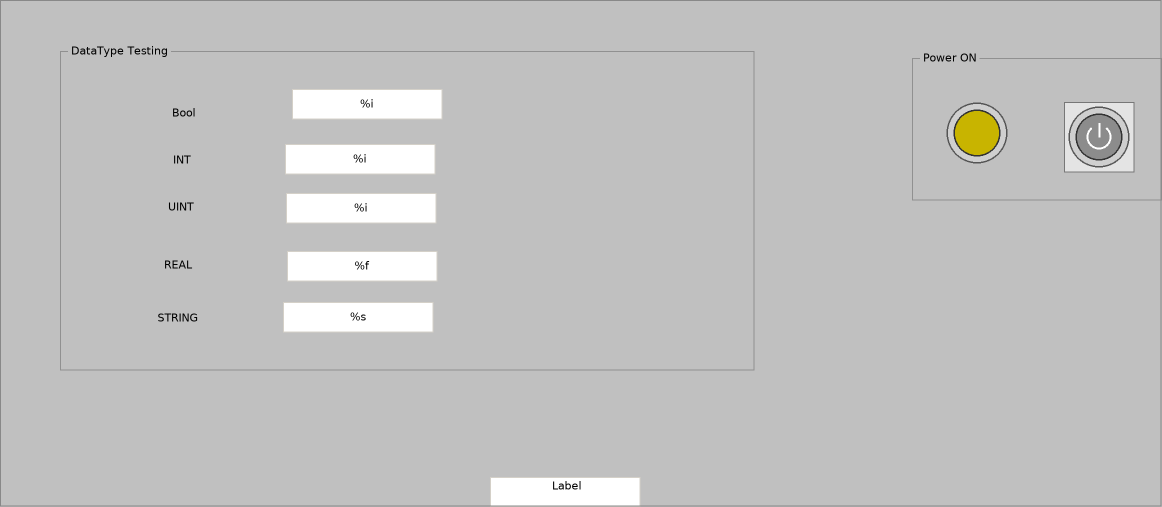
VISUALIZATION HMI  // 1162x507
    GroupBox (912,50 250x150), "Power ON"
        Lamp1 (30,48 70x70), variable: MAIN.bEnable, style: Lamp-Lamp1-Yellow
        PowerSwitch (152,52 70x70), variable: MAIN.bStart, behaviour: TOGGLE, style: Switch-PowerSwitch-Gray
    GroupBox (60,43 694x327), "DataType Testing"
        Textfield (223,259 150x30), "%s", text variable: MAIN.sPowerStatus
            OnMouseDown: write the text variable via Default
        Textfield (232,46 150x30), "%i", text variable: MAIN.bEnable
        Textfield (225,101 150x30), "%i", text variable: MAIN.nINT
        Textfield (226,150 150x30), "%i", text variable: MAIN.nUINT
        Textfield (227,208 150x30), "%f", text variable: MAIN.fREAL
        Label (49,55 150x30), "Bool"
        Label (47,102 150x30), "INT"
        Label (46,149 150x30), "UINT"
        Label (43,207 150x30), "REAL"
        Label (43,260 150x30), "STRING"
    Textfield (490,477 150x30)
    Label (492,471 150x30), "Label"
END_VISUALIZATION

(* stored: Version 1.1.0.1, ProductVersion 3.1.4024.12
   Visu HMI: Id {a1a1e5df-2f48-44e4-9c0b-8a596b764d5e} *)
